VISUALIZATION Vertical_Arm_Traveling_Zone  // 2x2
END_VISUALIZATION

(* stored: Version 1.1.0.1, ProductVersion 3.1.4024.12
   Visu Vertical_Arm_Traveling_Zone: Id {d7f2b557-99a4-4129-bb83-3ccfd6bc3ce6} *)
